// TIA Portal V16 export
// export: Created 2022-09-01T14:29:21.16046Z, ExportSetting WithDefaults, DisplayName Totally Integrated Automation Portal, DisplayVersion V16, DisplayName TIA Portal Version Control Interface, DisplayVersion V16, DisplayName TIA Portal Openness, DisplayVersion V16, DisplayName STEP 7 Professional, DisplayVersion V16, DisplayName STEP 7 Safety, DisplayVersion V16, DisplayName WinCC Advanced, DisplayVersion V16
DATA_BLOCK "Etapas_Grafcet_1"   // DB4
{ S7_Optimized_Access := 'TRUE' }
VERSION : 0.1
// stored: AutoNumber true, IsOnlyStoredInLoadMemory false, IsRetainMemResEnabled false, IsWriteProtectedInAS false, MemoryReserve 100
   VAR RETAIN
      ETAPA_1 : Bool;
      ETAPA_2 : Bool;
      ETAPA_3 : Bool;
      ETAPA_4 : Bool;
      ETAPA_5 : Bool;
      ETAPA_6 : Bool;
      ETAPA_7 : Bool;
      ETAPA_8 : Bool;
      ETAPA_9 : Bool;
      ETAPA_33 : Bool;
      ETAPA_55 : Bool;
      RESET_ETAPA_1 : Bool;
      SUSPENSÃO_CICLO : Bool;
   END_VAR
BEGIN
END_DATA_BLOCK
